Staubli VAL3: interfaceCS8.dtx

mdesc mNomSpeed
screen scMonitor
